// TIA Portal V19 export
FUNCTION "ItemControlMain" : Void   // FC49, STL
TITLE = Item main control
{ S7_Optimized_Access := 'TRUE' }
AUTHOR : FLA
FAMILY : UHT
VERSION : 1.0
// Item main control
// 
// Programmer Init: 8953-FLA
// 
// Change Log:
// 
// Date        Change                          Updated by
// ------------------------------------------------------
// 19.04.99    1. Edition                      FLA
// stored: AutoNumber false
BEGIN

NETWORK
TITLE = Service off all items
      L     "TRIGGERBYTE";  // Load trigger byte
      SLW   1;  // Shift to next trigger bit
      T     "TRIGGERBYTE";  // Save in trigger byte
      A     "T20_Trigger_bit";
      JC    L1;  // Timer running
      S     "Trigger bit 1";  // Set trigger 1

      CALL  "StartTimer"
      ( TIME_IN_SECONDS := 1,  // Time in seconds
        _TIMER          := "T20_Trigger_bit"  // Timer number
      );  // Start timer

L1:   NOP   0;

      A     "Trigger bit 1";  // Trigger bit 1
      =     "1hz_oneshot_valve handle";  // 1Hz oneshot
      CALL  "ControlAutobit1";  // Service items Q 32.0 to Q 45.7
      CALL  "OutputHandler1";

      A     "Trigger bit 2";  // Trigger bit 2
      =     "1hz_oneshot_valve handle";  // 1Hz oneshot
      CALL  "ControlAutobit2";  // Service items Q 64.0 to Q 77.7
      CALL  "OutputHandler2";

      A     "Trigger bit 3";
      =     "1hz_oneshot_valve handle";  // 1Hz oneshot
      CALL  "ControlAutoBit3";  // Service items
      CALL  "OutputHandler3";



NETWORK
TITLE = Update inputs to Intouch
// DB 16 used by Intouch
      L     "Tag_82";
      T     "InputsToScada".dw0;

      L     "Tag_83";
      T     "InputsToScada".dw2;

      L     "Tag_84";
      T     "InputsToScada".dw4;

      L     "Tag_85";
      T     "InputsToScada".dw6;

      L     "Tag_86";
      T     "InputsToScada".dw8;

      L     "Tag_87";
      T     "InputsToScada".dw10;

END_FUNCTION
